FUNCTION_BLOCK ArgoRx (* goFB_ignore *)
  (* Standard: 61499-2 *)
  (* Version 0.1, 2017-00-09, hpea485, UOA *)
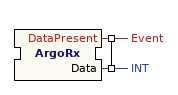
  EVENT_OUTPUT
    DataPresent WITH Data;
  END_EVENT
  VAR_OUTPUT
    Data : INT;
  END_VAR
  EC_STATES
    Start;
  END_STATES
END_FUNCTION_BLOCK
